// TwinCAT 3 PLC project opdracht
// ProgramVersion: 3.1.4023.0
// libraries:
//   Tc2_BABasic, * (Beckhoff Automation GmbH)
//   Tc2_LON, * (Beckhoff Automation GmbH)
//   Tc2_Standard, * (Beckhoff Automation GmbH)
//   Tc2_System, * (Beckhoff Automation GmbH)
//   Tc2_Utilities, * (Beckhoff Automation GmbH)
//   Tc3_IotBase, * (Beckhoff Automation GmbH)
//   Tc3_JsonXml, * (Beckhoff Automation GmbH)
//   Tc3_LS, * (Beckhoff Automation GmbH)
//   Tc3_Module, * (Beckhoff Automation GmbH)
//   VisuDialogs, * (System)
// project tree:
//   / GlobalTextList.TcGTLO, PlcTask.TcTTO, Visualization Manager.TcVMO (not stored)
//   GVLs/ GVL.TcGVL
//   POUs/ csvwrite.TcPOU, MAIN.TcPOU, Kamers.TcDUT, MQTT.TcPOU, terras1.TcDUT
//   POUs/OpenWeatherMap/ FB_TestHTTP_Get_openWeatherMapLat.TcPOU
//   VISUs/ Visualization.TcVIS

CONFIGURATION opdracht
    RESOURCE PLC ON TwinCAT3
        TASK PlcTask(INTERVAL := T#10ms, PRIORITY := 20);
        PROGRAM MAIN WITH PlcTask : MAIN;
    END_RESOURCE
END_CONFIGURATION

// ---- POUs/Kamers.TcDUT
TYPE Kamers :
STRUCT
	Lamp1 : BOOL;
	schakelaar : BOOL;	
	tempValue : INT := 21;
	lightToggle : FB_Light;
	chauffage : bool;
END_STRUCT
END_TYPE

// ---- POUs/terras1.TcDUT
TYPE terras1 EXTENDS Kamers :
STRUCT
watersproeier : BOOL;	

END_STRUCT
END_TYPE

// ---- GVLs/GVL.TcGVL
VAR_GLOBAL CONSTANT
	MAX_CSV_ROWS 			: UDINT := 100;
	MAX_CSV_COLUMNS 		: UDINT := 5;
	MAX_CSV_FIELD_LENGTH	: UDINT := 100;
	
	autorefresh : BOOL;
	
END_VAR

VAR_GLOBAL
	var1: INT;
END_VAR

// ---- POUs/MAIN.TcPOU
PROGRAM MAIN
VAR

	
	slaapkamerLamp2 : BOOL;
	ingesteldeTemp : INT := 20;
	temp : BOOL;
	chauffageOn : bool;
	
	living : kamers;
	wc : Kamers;
	keuken : Kamers;	
	terras : terras1;
	
	csvOpen : FB_FileOpen;	
	bGetOpenWeatherMap 				: BOOL;
	fbHttpClientOpenWeatherMap		: FB_IotHttpClient :=(sHostName:='api.openweathermap.org',
								  	bKeepAlive:=TRUE,	tConnectionTimeout:=T#10S);	
	GetValues			: FB_TestHTTP_Get_openWeatherMapLat;
	
	logs : BOOL := FALSE;
    trig : R_TRIG;
	chaufageTrig : R_trig;
	toggleEvent: BOOL;
	temptrigger : ton;

	
END_VAR
VAR_INPUT
	slaapkamer1 : Kamers;
	slaapkamer2 : Kamers;
END_VAR

//init client parameters at startup
// init client parameters at startup
temptrigger(in := NOT temptrigger.q, pt := T#1M);
GetTemp();
lights();
chauffage();
watersproeier();
csvwrite();
MQTT();
eventtest();

ACTION chauffage:

IF 	chauffageOn THEN 
	IF ( slaapkamer1.tempValue < (ingesteldeTemp -1))
			THEN
			slaapkamer1.chauffage := TRUE;
		ELSIF ( slaapkamer1.tempValue > (ingesteldeTemp + 1))
			THEN
			slaapkamer1.chauffage := FALSE;
		END_IF
		
		
	IF ( slaapkamer2.tempValue < (ingesteldeTemp -1))
			THEN
			slaapkamer2.chauffage := TRUE;
		ELSIF ( slaapkamer2.tempValue > (ingesteldeTemp + 1))
			THEN
			slaapkamer2.chauffage := FALSE;
		END_IF
		
	IF ( wc.tempValue < (ingesteldeTemp -1))
			THEN
			wc.chauffage := TRUE;
		ELSIF ( wc.tempValue > (ingesteldeTemp + 1))
			THEN
			wc.chauffage := FALSE;
		END_IF
		
	IF ( living.tempValue < (ingesteldeTemp -1))
			THEN
			living.chauffage := TRUE;
		ELSIF ( living.tempValue > (ingesteldeTemp + 1))
			THEN
			living.chauffage := FALSE;
		END_IF
		
	IF ( keuken.tempValue < (ingesteldeTemp -1))
			THEN
		keuken.chauffage := TRUE;
	ELSIF ( keuken.tempValue > (ingesteldeTemp + 1))
		THEN
		keuken.chauffage := FALSE;
	END_IF
ELSE
 	keuken.chauffage := FALSE;
	slaapkamer1.chauffage := FALSE;
	slaapkamer2.chauffage := FALSE;
	wc.chauffage := FALSE;
	living.chauffage := FALSE;
END_IF
END_ACTION

ACTION EventTest:
trig(clk := toggleEvent);
IF slaapkamer1.schakelaar THEN 
	var1 := 4;
	toggleEvent := TRUE;
ELSIF slaapkamer2.schakelaar THEN 
	var1 := 5;
	toggleEvent := TRUE;
ELSIF living.schakelaar THEN 
	var1 := 3;
	toggleEvent := TRUE;
ELSIF wc.schakelaar THEN 
	var1 := 1;
	toggleEvent := TRUE;
ELSIF terras.schakelaar THEN 
	var1 := 6;
	toggleEvent := TRUE;
ELSIF keuken.schakelaar THEN 
	var1 := 2;
	toggleEvent := TRUE;
ELSE
	toggleevent := FALSE;
END_IF
END_ACTION

ACTION GetTemp:
IF NOT fbHttpClientOpenWeatherMap.bConfigured THEN 
	fbHttpClientOpenWeatherMap.nHostPort:= 443;
	fbHttpClientOpenWeatherMap.stTLS.bNoServerCertCheck:= TRUE;
END_IF

IF fbHttpClientOpenWeatherMap.bConfigured THEN
	GetValues(bSend:=bGetOpenWeatherMap, fbClient:=fbHttpClientOpenWeatherMap);
 	
END_IF

fbHttpClientOpenWeatherMap.Execute();
END_ACTION

ACTION lights:
slaapkamer1.lightToggle( btoggle := slaapkamer1.schakelaar OR mqtt.fbtoggle1.Q , blight => slaapkamer1.Lamp1);
slaapkamer2.lightToggle( btoggle := slaapkamer2.schakelaar OR mqtt.fbtoggle2.q , blight => slaapkamer2.Lamp1);
keuken.lightToggle( btoggle := keuken.schakelaar OR mqtt.fbtoggle3.q , blight => keuken.Lamp1);

wc.lightToggle( btoggle := wc.schakelaar OR mqtt.fbtoggle4.q , blight => wc.Lamp1);
living.lightToggle( btoggle := living.schakelaar OR mqtt.fbtoggle5.q , blight => living.Lamp1);
terras.lightToggle( btoggle := terras.schakelaar OR mqtt.fbtoggle6.q , blight => terras.Lamp1);
END_ACTION

ACTION watersproeier:
IF terras.tempValue > 25 THEN
	terras.watersproeier := TRUE;
ELSE 
	terras.watersproeier := FALSE;
END_IF
END_ACTION

END_PROGRAM

// ---- POUs/OpenWeatherMap/FB_TestHTTP_Get_openWeatherMapLat.TcPOU
FUNCTION_BLOCK FB_TestHTTP_Get_openWeatherMapLat
VAR_INPUT
	bSend				: BOOL;
END_VAR
VAR_IN_OUT
	fbClient			: FB_IotHttpClient;
END_VAR
VAR_OUTPUT
	bBusy				: BOOL;
	bError				: BOOL;
END_VAR
VAR
	fbRequest			: FB_IotHttpRequest;
	fbJson				: FB_JsonDomParser;
	nState				: UDINT;
	RisingEdge			: R_TRIG;
	city : STRING;
	getweather : STRING := '/data/2.5/weather?q=';
	getweather2 : STRING := ',BE&appid=6E741a8faaaf146476fd94ab87413c7b&units=metric';
	getWeatherTotal : STRING(300);
	
	timerweather : ton;
	bGetContentResult	: BOOL;
	sContent			: STRING(511);	
	
	bGetJsonResult		: BOOL;
	jsonDoc				: SJsonValue;
	jsonVal				: SJsonValue;
	sResultValue		: STRING;
	
	nReqCount			: UDINT;	
	nResCount			: UDINT;
	nValidResCount		: UDINT;
	nErrCount			: UDINT;
	addstring: STRING;
	jsonprop: SJsonValue;
	jsonserial: SJsonValue;
	sTemp: LREAL ;
	
END_VAR

RisingEdge(CLK:= bSend);
IF autorefresh THEN 
	timerweather(in := NOT timerweather.Q, PT := T#30S);
END_IF


CASE nState OF
0:	
	IF RisingEdge.Q  THEN 
		addstring := concat(city , getweather2);
		getweathertotal := concat(getweather , addstring);
		
		
		IF fbRequest.SendRequest(sUri:= getweathertotal , fbClient:=fbClient, eRequestType:=ETcIotHttpRequestType.HTTP_Get, 0, 0, 0) THEN				
			nState:= 1;
			nReqCount:= nReqCount+1;
			bBusy:= TRUE;
			bError:= FALSE;
		END_IF					
	END_IF
	IF  timerweather.Q THEN 
		
		
		IF fbRequest.SendRequest(sUri:= getweathertotal , fbClient:=fbClient, eRequestType:=ETcIotHttpRequestType.HTTP_Get, 0, 0, 0) THEN				
			nState:= 1;
			nReqCount:= nReqCount+1;
			bBusy:= TRUE;
			bError:= FALSE;
		END_IF					
	END_IF
1:
	IF NOT fbRequest.bBusy THEN
		bError:= TRUE;
		IF NOT fbRequest.bError THEN				 
			bGetContentResult:= fbRequest.GetContent(pContent:= ADR(sContent), nContentSize:= SIZEOF(sContent), bSetNullTermination:= TRUE);
			IF fbRequest.nStatusCode >= 200 AND fbRequest.nStatusCode < 300 THEN
				bGetJsonResult:= FALSE;
				jsonDoc:= fbRequest.GetJsonDomContent(fbJson);
				IF jsonDoc <> 0 THEN
					parsen(); // do something with the weather data
					nValidResCount:= nValidResCount+1;
					bError:= FALSE;					
				END_IF							
				nResCount:= nResCount+1;			
			END_IF
		END_IF
		nState:= 0;
		bBusy:= FALSE;
		IF bError THEN
			nErrCount:= nErrCount+1;
		END_IF
	END_IF  	
END_CASE

ACTION parsen:
jsonprop := fbJson.FindMember(jsonDoc,'main');
IF (jsonprop <> 0) THEN
	jsonserial := fbjson.FindMember(jsonprop, 'temp');
	sTemp := fbjson.GetDouble(jsonserial);	
END_IF
END_ACTION

END_FUNCTION_BLOCK

// ---- POUs/csvwrite.TcPOU
PROGRAM csvwrite
VAR
	bWrite			: BOOL := FALSE;(* Rising edge starts program execution *)
	sNetId			: T_AmsNetId := '';	(* TwinCAT system network address *)
	sFileName		: T_MaxString := 'C:\Users\Administrator\Desktop\Log.csv';(* CSV destination file path and name *)
	sCSVLine		: T_MaxString := '';(* Single CSV text line (row, record), we are using string as record buffer (your are able to see created fields) *)
	sCSVField		: T_MaxString := '';(* Single CSV field value (column, record field) *)
	bBusy			: BOOL;
	bError			: BOOL;
	nErrId			: UDINT;
	nRow	 		: INT 	:= 0;(* Row number (record) *)
	nColumn			: UDINT 	:= 0;(* Column number (record field) *)
	hFile			: UINT		:= 0;(* File handle of the source file *)
	step			: DWORD 	:= 0;
	fbFileOpen		: FB_FileOpen;(* Opens file *)
	fbFileClose		: FB_FileClose;(* Closes file *)
	fbFilePuts		: FB_FilePuts;(* Writes one record (line) *)
	fbWriter		: FB_CSVMemBufferWriter;(* Helper function block used to create CSV data bytes (single record line) *)
	database		: ARRAY[0..MAX_CSV_COLUMNS ] OF STRING(MAX_CSV_FIELD_LENGTH) :=[ (* Source PLC database *)
	INT_TO_STRING(nRow), INT_TO_STRING(main.keuken.tempValue), INT_TO_STRING(main.living.tempValue), INT_TO_STRING(main.wc.tempValue), INT_TO_STRING(main.slaapkamer1.tempValue), INT_TO_STRING(main.slaapkamer2.tempValue)];
	ColumnNames : ARRAY[0..Max_CSV_COLUMNS] OF STRING(MAX_CSV_FIELD_LENGTH) := ['NR', 'TempKeuken', 'TempLiving', 'TempWC', 'TempSlaapkamer1', 'TempSlaapkamer2'  ];

END_VAR

CASE step OF
	0:	(* Wait for rising edge at bWrite variable *)
		IF main.temptrigger.q THEN
			bWrite 	:= FALSE;
			bBusy 	:= TRUE;
			bError	:= FALSE;
			nErrId	:= 0;
			hFile	:= 0;
			//nRow	:= 0;
			nColumn	:= 0;
			step 	:= 1;
			database[0]:=INT_TO_STRING(nRow);
			database[1]:=INT_TO_STRING(main.keuken.tempValue);
			database[2]:=INT_TO_STRING(main.living.tempValue);
			database[3]:=INT_TO_STRING(main.wc.tempValue);
			database[4]:=INT_TO_STRING(main.slaapkamer1.tempValue);
			database[5]:=INT_TO_STRING(main.slaapkamer2.tempValue);
			
		END_IF

	1:	(* Open source file *)
		fbFileOpen(  bExecute := FALSE  );
		fbFileOpen( sNetId := sNetId, sPathName := sFileName, nMode := FOPEN_MODEAPPEND OR FOPEN_MODETEXT,(* Open file in TEXT mode! *)
					ePath := PATH_GENERIC, bExecute := TRUE );
		step := 2;

	2:(* Wait until open not busy *)
		fbFileOpen( bExecute := FALSE, bError => bError, nErrID => nErrID, hFile => hFile );
		IF NOT fbFileOpen.bBusy THEN
			IF NOT fbFileOpen.bError THEN
				step := 3;
			ELSE(* Error: file not found? *)
				step := 100;
			END_IF
		END_IF

		
		
		
		
		
	3:(* Convert one PLC record to CSV format *)
		sCSVLine := '';
		fbWriter.eCmd := eEnumCmd_First;(* Write first field value *)
		

			FOR nColumn := 0 TO MAX_CSV_COLUMNS BY 1 DO

				sCSVField := STRING_TO_CSVFIELD( database[nColumn ], FALSE );(* TODO: Get field value from your application *)

				(* Add new field to the record buffer *)
				fbWriter( 	pBuffer := ADR( sCSVLine ), cbBuffer := SIZEOF( sCSVLine ) - 1, putValue := sCSVField, pValue := 0, cbValue := 0,
							bCRLF := ( nColumn = MAX_CSV_COLUMNS ) );(* bCRLF == TRUE => Write CRLF after the last field value *)
				IF fbWriter.bOk THEN
					fbWriter.eCmd := eEnumCmd_Next;(* Write next field value *)
				ELSE(* Error *)
					step := 100;
					RETURN;
				END_IF

			END_FOR(* FOR nColumn := 0... *)

			(* FB_FilePuts adds allready CR (carriage return) to the written line.
			We have to replace the $R$L characters with $L character to avoid double CR. *)
			IF RIGHT( sCSVLine, 2 ) = '$R$L' THEN
				sCSVLine := REPLACE( sCSVLine, '$L', 2, LEN( sCSVLine ) - 1 );
			END_IF

			nRow := nRow + 1;(* Increment number of created records (rows) *)
			step := 4;(* Write record to the file *)

		
			
		

	4:	(* Write single text line *)
		fbFilePuts( bExecute := FALSE );
		fbFilePuts( sNetId := sNetId, hFile := hFile, sLine := sCSVLine, bExecute := TRUE );
		step := 5;
		
		
		
		
		
		
		
		
		
		
		

	5:(* Wait until write not busy *)
		fbFilePuts( bExecute := FALSE, bError => bError, nErrID => nErrID );
		IF NOT fbFilePuts.bBusy THEN
			IF NOT fbFilePuts.bError THEN
				step := 10;(* Write next record *)
			ELSE(* Error *)
				step := 100;
			END_IF
		END_IF

		
		
		
		
		
		
		
		
		
		
		
	10:	(* Close source file *)
		fbFileClose( bExecute := FALSE );
		fbFileClose( sNetId := sNetId, hFile := hFile, bExecute := TRUE );
		step := 11;

	11:(* Wait until close not busy *)
		fbFileClose( bExecute := FALSE, bError => bError, nErrID => nErrID );
		IF ( NOT fbFileClose.bBusy ) THEN
			hFile := 0;
			step := 100;
		END_IF

	100: (* Error or ready step => cleanup *)
		IF ( hFile <> 0 ) THEN
			step := 10; (* Close the source file *)
		ELSE
			bBusy := FALSE;
			step := 0;	(* Ready *)
		END_IF

END_CASE

END_PROGRAM

// ---- POUs/MQTT.TcPOU
PROGRAM MQTT

VAR
	fbMqttClient : FB_IotMqttClient;
	bSetParameter : BOOL := TRUE;
	bConnect : BOOL := TRUE;
	
	(* published message *)
	sTopicPubTERRAS : STRING(255) := 'ToonBA?>TERRAS';
	sTopicPubWC: STRING(255) := 'ToonBA?>WC';
	sTopicPubLIVING : STRING(255) := 'ToonBA?>LIVING';
	sTopicPubSLAAPKAMER1 : STRING(255) := 'ToonBA?>SLAAPKAMER1';
	sTopicPubSLAAPKAMER2 : STRING(255) := 'ToonBA?>SLAAPKAMER2';
	sTopicPubKEUKEN : STRING(255) := 'ToonBA?>KEUKEN';
	sTopicPubTEMP : STRING(255) := 'ToonBA?>TEMP';
	
	sPayloadPub : STRING(255);
	i: UDINT;
	fbTimer : TON;
	
	sendbutton : BOOL;
	startbutton : BOOL;
	(* received message *)
	
	
	{attribute 'TcEncoding':='UTF-8'}
	sTopicRcv : STRING(255);
	{attribute 'TcEncoding':='UTF-8'}
	sPayloadRcv : STRING(255);
	fbMessageQueue : FB_IotMqttMessageQueue;
	fbMessage : FB_IotMqttMessage;
	trigger : R_TRIG;

	
	
	hrErrorOccurred : HRESULT; // contains the latest occurred error
	valueMQTT: STRING(255);
	sPayloadPubWC: STRING(255);
	sPayloadPubTERRAS: STRING(255);
	sPayloadPubKEUKEN: STRING(255);
	sPayloadPubLIVING: STRING(255);
	sPayloadPubSLAAPKAMER1: STRING(255);
	sPayloadPubSLAAPKAMER2: STRING(255);
	sPayloadPubWC1: STRING(255);
	sPayloadPubWC2: STRING(255);
	sPayloadPubWC3: STRING(255);
	l: INT;
	bSubscribed : BOOL;
	bSubscribed2: BOOL;
	bSubscribed3: BOOL;
	bSubscribed4: BOOL;
	bSubscribed5: BOOL;
	bSubscribed6: BOOL;
	sTopicSub1 : STRING(255) := 'ToonBA!>SLAAPKAMER1';
	sTopicSub2 : STRING(255) := 'ToonBA!>SLAAPKAMER2';
	sTopicSub3 : STRING(255) := 'ToonBA!>KEUKEN';
	sTopicSub4 : STRING(255) := 'ToonBA!>WC';
	sTopicSub5 : STRING(255) := 'ToonBA!>LIVING';
	sTopicSub6 : STRING(255) := 'ToonBA!>TERRAS';
	toggle : STRING(6) := 'toggle';
	toggle1: BOOL;
	toggle2: BOOL;
	toggle3: BOOL;
	toggle4: BOOL;
	toggle5: BOOL;
	toggle6: BOOL;
	fbtoggle1 : TP;
	fbtoggle2 : TP;
	fbtoggle3 : TP;
	fbtoggle4 : TP;
	fbtoggle5 : TP;
	fbtoggle6 : TP;

	sPayloadPubTEMP: STRING(255);
END_VAR

trigger( CLK := sendbutton);

ToggleV();
IF main.logs THEN
	fbtimer(in := NOT fbtimer.q,PT:=T#1M);
END_IF


IF bSetParameter THEN
	bSetParameter := FALSE;
	fbMqttClient.sHostName:= 'broker.mqttdashboard.com';
	fbMqttClient.nHostPort:= 1883;
//	fbMqttClient.sClientId:= 'ToonBACLIENT'; 
//	fbMqttClient.sTopicPrefix:= 'ToonBA?'; 
//	fbMqttClient.nKeepAlive:= 60; 
//	fbMqttClient.sUserName:= ;
//	fbMqttClient.sUserPassword:= ; 
//	fbMqttClient.stWill:= ; 
//	fbMqttClient.stTLS:= ;
	fbMqttClient.ipMessageQueue := fbMessageQueue;
END_IF

fbMqttClient.Execute(startbutton);
IF fbMqttClient.bError THEN
	// add your error logging here
	hrErrorOccurred := fbMqttClient.hrErrorCode;
END_IF

IF fbMessageQueue.nQueuedMessages > 0 THEN
	IF fbMessageQueue.Dequeue(fbMessage:=fbMessage) THEN
		fbMessage.GetTopic(pTopic:=ADR(sTopicRcv), nTopicSize:=SIZEOF(sTopicRcv) );
		fbMessage.GetPayload(pPayload:=ADR(sPayloadRcv), nPayloadSize:=SIZEOF(sPayloadRcv), bSetNullTermination:=TRUE);
		
		togglelamps();
		
	
		
	END_IF
END_IF

IF fbMqttClient.bConnected THEN
	//subscribe to all the topics
	subscribe();

	IF  trigger.Q  OR fbTimer.q THEN
		sendtopics();
	END_IF
	IF main.temptrigger.q THEN
		sPayloadPubTEMP := concat(concat(concat(concat(concat(CONCAT('keuken : ', TO_STRING(main.keuken.tempValue)), CONCAT(', living : ', TO_STRING(main.living.tempvalue))),CONCAT(', wc : ', TO_STRING(main.wc.tempvalue))),CONCAT(', slaapkamer1 : ', TO_STRING(main.slaapkamer1.tempvalue))),CONCAT(', slaapkamer2 : ', TO_STRING(main.slaapkamer2.tempvalue))),CONCAT(', terras : ', TO_STRING(main.terras.tempvalue)));
		
		fbMqttClient.Publish(	sTopic:= sTopicPubtemp, 
								pPayload:= ADR(sPayloadPubTEMP), nPayloadSize:= LEN2(ADR(sPayloadPubTEMP)), 
								eQoS:= TcIotMqttQos.AtMostOnceDelivery, bRetain:= FALSE, bQueue:= FALSE );
		IF fbMqttClient.bError THEN
			// add your error logging here
			hrErrorOccurred := fbMqttClient.hrErrorCode;
		END_IF
	END_IF
	
	// trigger for events and send values from what room triggered event
	
	IF  main.trig.q THEN 
		
		
	IF var1 = 1 THEN
		// SEND WC DATA //
		// SEND WC DATA //
		sPayloadPubWC := concat(concat(CONCAT('CHAUFFAGE = ', TO_STRING(main.wc.chauffage)), CONCAT(', TEMP = ', TO_STRING(main.wc.tempvalue))),CONCAT(', LAMP1 = ', TO_STRING(main.wc.Lamp1)));
		
		fbMqttClient.Publish(	sTopic:= sTopicPubWC, 
								pPayload:= ADR(sPayloadPubWC), nPayloadSize:= LEN2(ADR(sPayloadPubWC)), 
								eQoS:= TcIotMqttQos.AtMostOnceDelivery, bRetain:= FALSE, bQueue:= FALSE );
		IF fbMqttClient.bError THEN
			// add your error logging here
			hrErrorOccurred := fbMqttClient.hrErrorCode;
		END_IF
	ELSIF var1 = 2 THEN
		// SEND KEUKEN DATA //
			// SEND KEUKEN DATA //
			sPayloadPubKEUKEN := concat(concat(CONCAT('CHAUFFAGE = ', TO_STRING(main.KEUKEN.chauffage)), CONCAT(', TEMP = ', TO_STRING(main.KEUKEN.tempvalue))),CONCAT(', LAMP1 = ', TO_STRING(main.KEUKEN.Lamp1)));
			
			fbMqttClient.Publish(	sTopic:= sTopicPubKEUKEN, 
									pPayload:= ADR(sPayloadPubKEUKEN), nPayloadSize:= LEN2(ADR(sPayloadPubKEUKEN)), 
									eQoS:= TcIotMqttQos.AtMostOnceDelivery, bRetain:= FALSE, bQueue:= FALSE );
			IF fbMqttClient.bError THEN
				// add your error logging here
				hrErrorOccurred := fbMqttClient.hrErrorCode;
			END_IF
		
	ELSIF var1 = 3 THEN
		// SEND LIVING DATA //
			// SEND LIVING DATA //
			sPayloadPubLIVING := concat(concat(CONCAT('CHAUFFAGE = ', TO_STRING(main.LIVING.chauffage)), CONCAT(', TEMP = ', TO_STRING(main.LIVING.tempvalue))),CONCAT(', LAMP1 = ', TO_STRING(main.LIVING.Lamp1)));
			
			fbMqttClient.Publish(	sTopic:= sTopicPubLIVING, 
									pPayload:= ADR(sPayloadPubLIVING), nPayloadSize:= LEN2(ADR(sPayloadPubLIVING)), 
									eQoS:= TcIotMqttQos.AtMostOnceDelivery, bRetain:= FALSE, bQueue:= FALSE );
			IF fbMqttClient.bError THEN
				// add your error logging here
				hrErrorOccurred := fbMqttClient.hrErrorCode;
			END_IF
		
	ELSIF var1 = 4 THEN
		// SEND SLAAPKAMER1 DATA //
			// SEND SLAAPKAMER1 DATA //
			
			
			sPayloadPubSLAAPKAMER1 := concat(concat(CONCAT('CHAUFFAGE = ', TO_STRING(main.SLAAPKAMER1.chauffage)), CONCAT(', TEMP = ', TO_STRING(main.SLAAPKAMER1.tempvalue))),CONCAT(', LAMP1 = ', TO_STRING(main.SLAAPKAMER1.Lamp1)));
			
			fbMqttClient.Publish(	sTopic:= sTopicPubSLAAPKAMER1, 
									pPayload:= ADR(sPayloadPubSLAAPKAMER1), nPayloadSize:= LEN2(ADR(sPayloadPubSLAAPKAMER1)), 
									eQoS:= TcIotMqttQos.AtMostOnceDelivery, bRetain:= FALSE, bQueue:= FALSE );
			IF fbMqttClient.bError THEN
				// add your error logging here
				hrErrorOccurred := fbMqttClient.hrErrorCode;
			END_IF
	ELSIF var1 = 5 THEN
		// SEND SLAAPKAMER2 DATA //
			// SEND SLAAPKAMER2 DATA //
			
			
			sPayloadPubSLAAPKAMER2 := concat(concat(CONCAT('CHAUFFAGE = ', TO_STRING(main.SLAAPKAMER2.chauffage)), CONCAT(', TEMP = ', TO_STRING(main.SLAAPKAMER2.tempvalue))),CONCAT(', LAMP1 = ', TO_STRING(main.SLAAPKAMER2.Lamp1)));
			
			fbMqttClient.Publish(	sTopic:= sTopicPubSLAAPKAMER2, 
									pPayload:= ADR(sPayloadPubSLAAPKAMER2), nPayloadSize:= LEN2(ADR(sPayloadPubSLAAPKAMER2)), 
									eQoS:= TcIotMqttQos.AtMostOnceDelivery, bRetain:= FALSE, bQueue:= FALSE );
			IF fbMqttClient.bError THEN
				// add your error logging here
				hrErrorOccurred := fbMqttClient.hrErrorCode;
			END_IF
		
	ELSIF var1 = 6 THEN	
		// SEND TERRAS DATA //
			// SEND TERRAS DATA //
			
			
			sPayloadPubTERRAS := concat(concat(CONCAT('watersproeier = ', TO_STRING(main.TERRAS.watersproeier)), CONCAT(', TEMP = ', TO_STRING(main.TERRAS.tempvalue))),CONCAT(', LAMP1 = ', TO_STRING(main.TERRAS.Lamp1)));
			
			fbMqttClient.Publish(	sTopic:= sTopicPubTERRAS, 
									pPayload:= ADR(sPayloadPubTERRAS), nPayloadSize:= LEN2(ADR(sPayloadPubTERRAS)), 
									eQoS:= TcIotMqttQos.AtMostOnceDelivery, bRetain:= FALSE, bQueue:= FALSE );
			IF fbMqttClient.bError THEN
				// add your error logging here
				hrErrorOccurred := fbMqttClient.hrErrorCode;
			END_IF
		
		
		
		
END_IF
	END_IF
END_IF

ACTION sendtopics:
	
		// SEND WC DATA //
		// SEND WC DATA //
		sPayloadPubWC := concat(concat(CONCAT('CHAUFFAGE = ', TO_STRING(main.wc.chauffage)), CONCAT(', TEMP = ', TO_STRING(main.wc.tempvalue))),CONCAT(', LAMP1 = ', TO_STRING(main.wc.Lamp1)));
		
		fbMqttClient.Publish(	sTopic:= sTopicPubWC, 
								pPayload:= ADR(sPayloadPubWC), nPayloadSize:= LEN2(ADR(sPayloadPubWC)), 
								eQoS:= TcIotMqttQos.AtMostOnceDelivery, bRetain:= FALSE, bQueue:= FALSE );
		IF fbMqttClient.bError THEN
			// add your error logging here
			hrErrorOccurred := fbMqttClient.hrErrorCode;
		END_IF
		
		// SEND KEUKEN DATA //
		// SEND KEUKEN DATA //
		sPayloadPubKEUKEN := concat(concat(CONCAT('CHAUFFAGE = ', TO_STRING(main.KEUKEN.chauffage)), CONCAT(', TEMP = ', TO_STRING(main.KEUKEN.tempvalue))),CONCAT(', LAMP1 = ', TO_STRING(main.KEUKEN.Lamp1)));
		
		fbMqttClient.Publish(	sTopic:= sTopicPubKEUKEN, 
								pPayload:= ADR(sPayloadPubKEUKEN), nPayloadSize:= LEN2(ADR(sPayloadPubKEUKEN)), 
								eQoS:= TcIotMqttQos.AtMostOnceDelivery, bRetain:= FALSE, bQueue:= FALSE );
		IF fbMqttClient.bError THEN
			// add your error logging here
			hrErrorOccurred := fbMqttClient.hrErrorCode;
		END_IF
		// SEND LIVING DATA //
		// SEND LIVING DATA //
		sPayloadPubLIVING := concat(concat(CONCAT('CHAUFFAGE = ', TO_STRING(main.LIVING.chauffage)), CONCAT(', TEMP = ', TO_STRING(main.LIVING.tempvalue))),CONCAT(', LAMP1 = ', TO_STRING(main.LIVING.Lamp1)));
		
		fbMqttClient.Publish(	sTopic:= sTopicPubLIVING, 
								pPayload:= ADR(sPayloadPubLIVING), nPayloadSize:= LEN2(ADR(sPayloadPubLIVING)), 
								eQoS:= TcIotMqttQos.AtMostOnceDelivery, bRetain:= FALSE, bQueue:= FALSE );
		IF fbMqttClient.bError THEN
			// add your error logging here
			hrErrorOccurred := fbMqttClient.hrErrorCode;
		END_IF
		
		// SEND SLAAPKAMER1 DATA //
		// SEND SLAAPKAMER1 DATA //
		
		
		sPayloadPubSLAAPKAMER1 := concat(concat(CONCAT('CHAUFFAGE = ', TO_STRING(main.SLAAPKAMER1.chauffage)), CONCAT(', TEMP = ', TO_STRING(main.SLAAPKAMER1.tempvalue))),CONCAT(', LAMP1 = ', TO_STRING(main.SLAAPKAMER1.Lamp1)));
		
		fbMqttClient.Publish(	sTopic:= sTopicPubSLAAPKAMER1, 
								pPayload:= ADR(sPayloadPubSLAAPKAMER1), nPayloadSize:= LEN2(ADR(sPayloadPubSLAAPKAMER1)), 
								eQoS:= TcIotMqttQos.AtMostOnceDelivery, bRetain:= FALSE, bQueue:= FALSE );
		IF fbMqttClient.bError THEN
			// add your error logging here
			hrErrorOccurred := fbMqttClient.hrErrorCode;
		END_IF
		
	
		
		// SEND SLAAPKAMER2 DATA //
		// SEND SLAAPKAMER2 DATA //
		
		
		sPayloadPubSLAAPKAMER2 := concat(concat(CONCAT('CHAUFFAGE = ', TO_STRING(main.SLAAPKAMER2.chauffage)), CONCAT(', TEMP = ', TO_STRING(main.SLAAPKAMER2.tempvalue))),CONCAT(', LAMP1 = ', TO_STRING(main.SLAAPKAMER2.Lamp1)));
		
		fbMqttClient.Publish(	sTopic:= sTopicPubSLAAPKAMER2, 
								pPayload:= ADR(sPayloadPubSLAAPKAMER2), nPayloadSize:= LEN2(ADR(sPayloadPubSLAAPKAMER2)), 
								eQoS:= TcIotMqttQos.AtMostOnceDelivery, bRetain:= FALSE, bQueue:= FALSE );
		IF fbMqttClient.bError THEN
			// add your error logging here
			hrErrorOccurred := fbMqttClient.hrErrorCode;
		END_IF
		
		// SEND TERRAS DATA //
		// SEND TERRAS DATA //
		
		
		sPayloadPubTERRAS := concat(concat(CONCAT('watersproeier = ', TO_STRING(main.TERRAS.watersproeier)), CONCAT(', TEMP = ', TO_STRING(main.TERRAS.tempvalue))),CONCAT(', LAMP1 = ', TO_STRING(main.TERRAS.Lamp1)));
		
		fbMqttClient.Publish(	sTopic:= sTopicPubTERRAS, 
								pPayload:= ADR(sPayloadPubTERRAS), nPayloadSize:= LEN2(ADR(sPayloadPubTERRAS)), 
								eQoS:= TcIotMqttQos.AtMostOnceDelivery, bRetain:= FALSE, bQueue:= FALSE );
		IF fbMqttClient.bError THEN
			// add your error logging here
			hrErrorOccurred := fbMqttClient.hrErrorCode;
		END_IF
END_ACTION

ACTION Subscribe:
IF NOT bSubscribed THEN
		bSubscribed := fbMqttClient.Subscribe(sTopic:=sTopicSub1, eQoS:=TcIotMqttQos.AtMostOnceDelivery);
		IF fbMqttClient.bError THEN
			// add your error logging here
			hrErrorOccurred := fbMqttClient.hrErrorCode;
		END_IF
	END_IF
	IF NOT bSubscribed2 THEN
		bSubscribed2 := fbMqttClient.Subscribe(sTopic:=sTopicSub2, eQoS:=TcIotMqttQos.AtMostOnceDelivery);
		IF fbMqttClient.bError THEN
			// add your error logging here
			hrErrorOccurred := fbMqttClient.hrErrorCode;
		END_IF
	END_IF
	IF NOT bSubscribed3 THEN
		bSubscribed3 := fbMqttClient.Subscribe(sTopic:=sTopicSub3, eQoS:=TcIotMqttQos.AtMostOnceDelivery);
		IF fbMqttClient.bError THEN
			// add your error logging here
			hrErrorOccurred := fbMqttClient.hrErrorCode;
		END_IF
	END_IF
	IF NOT bSubscribed4 THEN
		bSubscribed4 := fbMqttClient.Subscribe(sTopic:=sTopicSub4, eQoS:=TcIotMqttQos.AtMostOnceDelivery);
		IF fbMqttClient.bError THEN
			// add your error logging here
			hrErrorOccurred := fbMqttClient.hrErrorCode;
		END_IF
	END_IF
	IF NOT bSubscribed5 THEN
		bSubscribed5 := fbMqttClient.Subscribe(sTopic:=sTopicSub5, eQoS:=TcIotMqttQos.AtMostOnceDelivery);
		IF fbMqttClient.bError THEN
			// add your error logging here
			hrErrorOccurred := fbMqttClient.hrErrorCode;
		END_IF
	END_IF
	IF NOT bSubscribed6 THEN
		bSubscribed6 := fbMqttClient.Subscribe(sTopic:=sTopicSub6, eQoS:=TcIotMqttQos.AtMostOnceDelivery);
		IF fbMqttClient.bError THEN
			// add your error logging here
			hrErrorOccurred := fbMqttClient.hrErrorCode;
		END_IF
	END_IF
END_ACTION

ACTION ToggleLamps:
IF sTopicRcv = sTopicSub1 THEN
			IF sPayloadRcv = toggle THEN				
					toggle1 := TRUE;					
			END_IF
		ELSIF sTopicRcv = sTopicSub2 THEN
			IF sPayloadRcv = toggle THEN				
					toggle2 := TRUE;					
			END_IF
		ELSIF sTopicRcv = sTopicSub3 THEN
			IF sPayloadRcv = toggle THEN				
					toggle3 := TRUE;					
			END_IF
		ELSIF sTopicRcv = sTopicSub4 THEN
			IF sPayloadRcv = toggle THEN				
					toggle4 := TRUE;					
			END_IF
		ELSIF sTopicRcv = sTopicSub5 THEN
			IF sPayloadRcv = toggle THEN				
					toggle5 := TRUE;					
			END_IF
		ELSIF sTopicRcv = sTopicSub6 THEN
			IF sPayloadRcv = toggle THEN				
					toggle6 := TRUE;					
			END_IF			
		END_IF
END_ACTION

ACTION ToggleV:
fbtoggle1(in := toggle1);
fbtoggle2(in := toggle2);
fbtoggle3(in := toggle3);
fbtoggle4(in := toggle4);
fbtoggle5(in := toggle5);
fbtoggle6(in := toggle6);
IF fbtoggle1.Q THEN 
	toggle1 := FALSE;
END_IF
IF fbtoggle2.Q THEN 
	toggle2 := FALSE;
END_IF
IF fbtoggle3.Q THEN 
	toggle3 := FALSE;
END_IF
IF fbtoggle4.Q THEN 
	toggle4 := FALSE;
END_IF
IF fbtoggle5.Q THEN 
	toggle5 := FALSE;
END_IF
IF fbtoggle6.Q THEN 
	toggle6 := FALSE;
END_IF
END_ACTION

END_PROGRAM

// ---- GlobalTextList.TcGTLO
TEXTLIST GlobalTextList
  177 = '%f'
  601 = '%s'
  166 = 'autoLog'
  94 = 'autorefresh'
  223 = 'Autorefresh'
  560 = 'AutoUpdate'
  77 = 'chauffage'
  287 = 'city:'
  840 = 'GetWeather'
  701 = 'keuken'
  839 = 'living'
  431 = 'send mqtt'
  419 = 'slaapkamer1'
  228 = 'slaapkamer2'
  706 = 'start mqtt'
  160 = 'temp sensors'
  377 = 'temp:'
  318 = 'temp: %d'
  472 = 'Terras'
  169 = 'watersproeier'
  675 = 'wc'
END_TEXTLIST

// ---- VISUs/Visualization.TcVIS
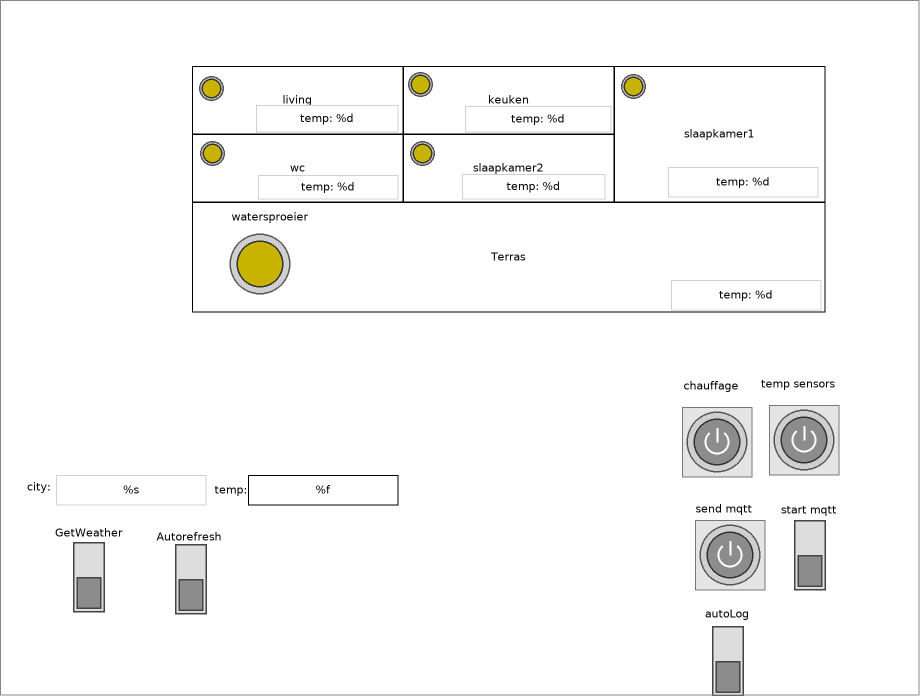
VISUALIZATION Visualization  // 920x696
    Rectangle (192,66 211x68), "living", colour toggle: MAIN.living.Lamp1
        tap MAIN.living.schakelaar
    Rectangle (403,66 211x68), "keuken", colour toggle: MAIN.keuken.Lamp1
        tap MAIN.keuken.schakelaar
    Rectangle (192,134 211x68), "wc", colour toggle: MAIN.wc.Lamp1
        tap MAIN.wc.schakelaar
    Rectangle (403,134 211x68), "slaapkamer2", colour toggle: MAIN.slaapkamer2.Lamp1
        tap MAIN.slaapkamer2.schakelaar
    Rectangle (614,66 211x136), "slaapkamer1", colour toggle: MAIN.slaapkamer1.Lamp1
        tap MAIN.slaapkamer1.schakelaar
    Textfield (668,167 150x30), "temp: %d", text variable: MAIN.slaapkamer1.tempValue, invisible if: not MAIN.temp
        OnMouseDown: write the text variable via Default
    Textfield (462,174 143x25), "temp: %d", text variable: MAIN.slaapkamer2.tempValue, invisible if: not MAIN.temp
        OnMouseDown: write the text variable via Default
    Textfield (465,106 146x26), "temp: %d", text variable: MAIN.keuken.tempValue, invisible if: not MAIN.temp
        OnMouseDown: write the text variable via Default
    Textfield (256,105 142x27), "temp: %d", text variable: MAIN.living.tempValue, invisible if: not MAIN.temp
        OnMouseDown: write the text variable via Default
    Textfield (258,175 140x24), "temp: %d", text variable: MAIN.wc.tempValue, invisible if: not MAIN.temp
        OnMouseDown: write the text variable via Default
    PowerSwitch (769,405 70x70), variable: MAIN.temp, behaviour: TOGGLE, style: Switch-PowerSwitch-Gray
    Rectangle (192,202 633x110), "Terras", colour toggle: MAIN.terras.Lamp1
        tap MAIN.terras.schakelaar
    Textfield (671,280 150x30), "temp: %d", text variable: MAIN.terras.tempValue, invisible if: not MAIN.temp
        OnMouseDown: write the text variable via Default
    Lamp1 (196,74 31x29), variable: MAIN.living.chauffage, style: Lamp-Lamp1-Yellow
    Lamp1 (197,139 31x29), variable: MAIN.wc.chauffage, style: Lamp-Lamp1-Yellow
    Lamp1 (405,70 31x29), variable: MAIN.keuken.chauffage, style: Lamp-Lamp1-Yellow
    Lamp1 (618,72 31x29), variable: MAIN.slaapkamer1.chauffage, style: Lamp-Lamp1-Yellow
    Lamp1 (407,139 31x29), variable: MAIN.slaapkamer2.chauffage, style: Lamp-Lamp1-Yellow
    Label (723,369 150x30), "temp sensors"
    PowerSwitch (682,407 70x70), variable: MAIN.chauffageOn, behaviour: TOGGLE, style: Switch-PowerSwitch-Gray
    DipSwitch (54,542 70x70), variable: MAIN.bGetOpenWeatherMap, behaviour: TOGGLE, style: Switch-DipSwitch-Gray
    Textfield (56,475 150x30), "%s", text variable: MAIN.GetValues.city
        OnMouseClick: write the text variable via Default
    Rectangle (248,475 150x30), "%f", text variable: MAIN.GetValues.sTemp
    Label (210,478 42x24), "temp:"
    Label (-36,472 150x30), "city:"
    DipSwitch (775,520 70x70), variable: MQTT.startbutton, behaviour: TOGGLE, style: Switch-DipSwitch-Gray
    PowerSwitch (695,520 70x70), variable: MQTT.sendbutton, behaviour: TAP, style: Switch-PowerSwitch-Gray
    Label (734,495 150x30), "start mqtt"
    Label (649,494 150x30), "send mqtt"
    Lamp1 (225,229 70x70), variable: main.terras.watersproeier, style: Lamp-Lamp1-Yellow
    Label (195,202 150x30), "watersproeier"
    DipSwitch (693,626 70x70), tooltip "autoLog", variable: MAIN.logs, behaviour: TOGGLE, style: Switch-DipSwitch-Gray
    Label (652,599 150x30), "autoLog"
    DipSwitch (156,544 70x70), tooltip "autorefresh", variable: autorefresh, behaviour: TOGGLE, style: Switch-DipSwitch-Gray
    Label (14,518 150x30), "GetWeather"
    Label (114,522 150x30), "Autorefresh"
    Label (636,371 150x30), "chauffage"
END_VISUALIZATION
